ABB RAPID module: linear_test.mod

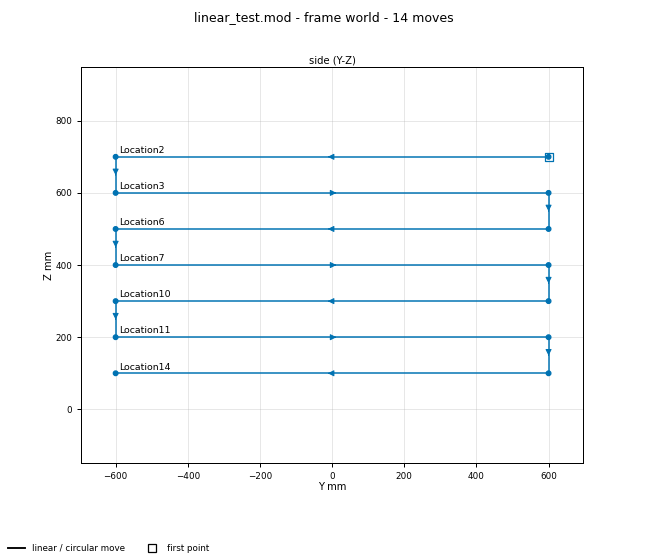
[picture p0: tool path of linear_test.mod in frame world, 14 of 14 moves have a stored position in this frame; points joined in program order, loops and branches not executed]
MODULE linear_test

    PERS robtarget Location1:=[[300, 600, 700], [0, 1, 0, 0], [-1, -1, 0, 1], [9000000000, 9000000000, 9000000000, 9000000000, 9000000000, 9000000000]];
    PERS robtarget Location2:=[[300, -600, 700], [0, 1, 0, 0], [-1, -1, 0, 1], [9000000000, 9000000000, 9000000000, 9000000000, 9000000000, 9000000000]];
    PERS robtarget Location3:=[[300, -600, 600], [0, 1, 0, 0], [-1, -1, 0, 1], [9000000000, 9000000000, 9000000000, 9000000000, 9000000000, 9000000000]];
    PERS robtarget Location4:=[[300, 600, 600], [0, 1, 0, 0], [-1, -1, 0, 1], [9000000000, 9000000000, 9000000000, 9000000000, 9000000000, 9000000000]];
    PERS robtarget Location5:=[[300, 600, 500], [0, 1, 0, 0], [-1, -1, 0, 1], [9000000000, 9000000000, 9000000000, 9000000000, 9000000000, 9000000000]];
    PERS robtarget Location6:=[[300, -600, 500], [0, 1, 0, 0], [-1, -1, 0, 1], [9000000000, 9000000000, 9000000000, 9000000000, 9000000000, 9000000000]];
    PERS robtarget Location7:=[[300, -600, 400], [0, 1, 0, 0], [-1, -1, 0, 1], [9000000000, 9000000000, 9000000000, 9000000000, 9000000000, 9000000000]];
    PERS robtarget Location8:=[[300, 600, 400], [0, 1, 0, 0], [-1, -1, 0, 1], [9000000000, 9000000000, 9000000000, 9000000000, 9000000000, 9000000000]];
    PERS robtarget Location9:=[[300, 600, 300], [0, 1, 0, 0], [-1, -1, 0, 1], [9000000000, 9000000000, 9000000000, 9000000000, 9000000000, 9000000000]];
    PERS robtarget Location10:=[[300, -600, 300], [0, 1, 0, 0], [-1, -1, 0, 1], [9000000000, 9000000000, 9000000000, 9000000000, 9000000000, 9000000000]];
    PERS robtarget Location11:=[[300, -600, 200], [0, 1, 0, 0], [-1, -1, 0, 1], [9000000000, 9000000000, 9000000000, 9000000000, 9000000000, 9000000000]];
    PERS robtarget Location12:=[[300, 600, 200], [0, 1, 0, 0], [-1, -1, 0, 1], [9000000000, 9000000000, 9000000000, 9000000000, 9000000000, 9000000000]];
    PERS robtarget Location13:=[[300, 600, 100], [0, 1, 0, 0], [-1, -1, 0, 1], [9000000000, 9000000000, 9000000000, 9000000000, 9000000000, 9000000000]];
    PERS robtarget Location14:=[[300, -600, 100], [0, 1, 0, 0], [-1, -1, 0, 1], [9000000000, 9000000000, 9000000000, 9000000000, 9000000000, 9000000000]];

	PROC main()
        ConfL\Off;
        MoveL Location1, v500, fine, tool0;
        MoveL Location2, v500, fine, tool0;
        MoveL Location3, v500, fine, tool0;
        MoveL Location4, v500, fine, tool0;
        MoveL Location5, v500, fine, tool0;
        MoveL Location6, v500, fine, tool0;
        MoveL Location7, v500, fine, tool0;
        MoveL Location8, v500, fine, tool0;
        MoveL Location9, v500, fine, tool0;
        MoveL Location10, v500, fine, tool0;
        MoveL Location11, v500, fine, tool0;
        MoveL Location12, v500, fine, tool0;
        MoveL Location13, v500, fine, tool0;
        MoveL Location14, v500, fine, tool0;
	ENDPROC

ENDMODULE
